TYPE ST_SysParameters :
STRUCT
	gen_SealAndPump				: STRING(100);
	cal_AcceptanceCriteria		: STRING(100);
	cal_AllowableFail			: STRING(100);
	cal_Replicates				: STRING(100);
	cal_PumpCallIntervalDays	: STRING(100);
	cal_CloseAppOnCompletation	: STRING(100);
	AirDryTimeOnCompletation	: STRING(100);
	lkt_AllowableLeakTestFail	: STRING(100);
	lkt_LeakTestBuildupTime		: STRING(100);
	lkt_LeakTestHoldTime		: STRING(100);
	lkt_LeakTestPressure		: STRING(100);
	mec_PlatesClosedPosition	: STRING(100);
	mec_PlatesDryPosition		: STRING(100);
	mec_PlatesVelocity			: STRING(100);
	mec_MaxCurrentFastDown		: STRING(100);
	mec_MaxCurrentSlowDown		: STRING(100);
	mec_MaxCurrentSlowUp		: STRING(100);
	pmp_MeterVelocity			: STRING(100);
	pmp_RunVelocity				: STRING(100);
	pmp_EmptyFactor				: STRING(100);
	pmp_FillSolventTubesFactor	: STRING(100);
	smp_AboveCalibration		: STRING(100);
	smp_VialSetSpacing			: STRING(100);
	smp_IntoResBottom			: STRING(100);
	smp_IntoResDispense			: STRING(100);
	smp_IntoResWeigh			: STRING(100);
	smp_IntoVials				: STRING(100);
	sec_DisplayManualControl	: STRING(100);
	sec_CheckLogonEachRun		: STRING(100);
	createdBy					: STRING(100);
	createdDate					: STRING(100);
	sysRevisionNo				: INT;
	
END_STRUCT
END_TYPE

(* stored: Version 1.1.0.1, ProductVersion 3.1.4024.15
   DUT ST_SysParameters: Id {5afcbe8d-8d8f-4737-8dcb-b0b24d2ad6bd} *)
